FUNCTION_BLOCK FB_ParseCommandOption
VAR
	sVersion: STRING:='0.9.0';
END_VAR
VAR_INPUT
	nCommandEndIndex:INT:=0;	
END_VAR
VAR
	psCommandBufferString: POINTER TO STRING; //string to point into byte buffer		
	nEqualSign: INT;
	nQuestionMark: INT;
END_VAR

VAR_IN_OUT
	byteCommandBuffer	:	ARRAY[0..PLCPRJ_BUFFER_SIZE] OF BYTE;//ADS input buffer
	nBytesInCommandBuffer:DINT:=0;
	nIndexEndOfCommand:DINT:=0;
END_VAR

VAR_OUTPUT
	nErrorId: UDINT;
	bError:BOOL:=FALSE;
	sSubErrorString: STRING;
	sStaticCommand:STRING;
	sStaticValue:STRING;
	bReadCommand:BOOL:=FALSE;
	bWriteCommand:BOOL:=FALSE;
	bWritePersistent:BOOL:=FALSE;	
END_VAR

//Parse static command	
nErrorId:=0;
bError:=FALSE;
sStaticCommand:='';
sStaticValue:='';
bReadCommand:=FALSE;
bWriteCommand:=FALSE;
bWritePersistent:=FALSE;		
psCommandBufferString:=ADR(byteCommandBuffer);

nEqualSign:=find(STR1:=PSTRING_TO_STRING(psCommandBufferString),STR2:=EPICS_WRITE_CMD);	
IF nEqualSign>0 AND nEqualSign<nCommandEndIndex THEN
	bWriteCommand:=TRUE;	
	//Command
	memcpy(destAddr:=ADR(sStaticCommand[0]),srcAddr:=ADR(byteCommandBuffer[0]),n:=nEqualSign-1);
	memset(destAddr	:=ADR(sStaticCommand[nEqualSign-1]),fillByte:=0,n:=1);				//Terminate string	
	//Check if persistent
	//IF find(STR1:=sStaticCommand,STR2:=EPICS_STATIC_COMMAND_PERSISTENT)>0 THEN
//		bWritePersistent:=TRUE;
//	END_IF
	//Value
	memcpy(destAddr:=ADR(sStaticValue[0]),srcAddr:=ADR(byteCommandBuffer[nEqualSign]),n:=nCommandEndIndex-nEqualSign-1);
	memset(destAddr	:=ADR(sStaticValue[nCommandEndIndex-nEqualSign-1]),fillByte:=0,n:=1); //Terminate string
	IF NOT F_RemoveBytesFromBuffer(nRemoveBytes:= nCommandEndIndex,byteCommandBuffer:=byteCommandBuffer,nBytesInCommandBuffer:=nBytesInCommandBuffer,nIndexEndOfCommand:=nIndexEndOfCommand) THEN 			
		bError:=TRUE;
		nErrorId:=301;
		sSubErrorString:='State 3: Failed to clear buffer (Parse static command write).';	
	END_IF				
ELSE
	nQuestionMark:=find(STR1:=PSTRING_TO_STRING(psCommandBufferString),STR2:=EPICS_READ_CMD);	
	IF nQuestionMark>0 AND nQuestionMark<nCommandEndIndex THEN
		bReadCommand:=TRUE;	
		//Command
		memcpy(destAddr:=ADR(sStaticCommand[0]),srcAddr:=ADR(byteCommandBuffer[0]),n:=nQuestionMark-1);
		memset(destAddr	:=ADR(sStaticCommand[nQuestionMark-1]),fillByte:=0,n:=1);				//Terminate string	

		//Clean buffer
		IF NOT F_RemoveBytesFromBuffer(nRemoveBytes:= nCommandEndIndex,byteCommandBuffer:=byteCommandBuffer,nBytesInCommandBuffer:=nBytesInCommandBuffer,nIndexEndOfCommand:=nIndexEndOfCommand) THEN 			
			bError:=TRUE;
			nErrorId:=302;
			sSubErrorString:='State 3: Failed to clear buffer (Parse static command read).';	
		END_IF		
	END_IF
END_IF	

IF NOT (bReadCommand OR  bWriteCommand) THEN										
	bError:=TRUE;
	nErrorId:=303;
	sSubErrorString:='State 3: Parsing of static command failed).';	
END_IF

END_FUNCTION_BLOCK

(* stored: Version 1.1.0.1, ProductVersion 3.1.0.25
   POU FB_ParseCommandOption: Id {1a6526d5-0082-4e55-944b-26a5f5166a94} *)
